PROGRAM StringHelper
VAR
END_VAR

// Converts the provided string to all lower case and returns the converted value.
METHOD ToLowerCase : T_MaxString
VAR_INPUT
	str	: Tc2_System.T_MaxString;	// Source string
END_VAR
ToLowerCase := Tc2_Utilities.F_ToLCase(in := str);
END_METHOD

// Converts the provided string to all upper case and returns the converted value.
METHOD ToUpperCase : Tc2_System.T_MaxString
VAR_INPUT
	str	: Tc2_System.T_MaxString;	// Source string
END_VAR
ToUpperCase := Tc2_Utilities.F_ToUCase(in := str);
END_METHOD

// Removes leading spaces from the character string and returns the reduced character string
METHOD PUBLIC TrimLeftSide : Tc2_System.T_MaxString
VAR_INPUT
	str	: Tc2_System.T_MaxString; // String to be trimmed
END_VAR
TrimRightSide := Tc2_Utilities.F_LTrim(in := str);
END_METHOD

// Truncates all trailing spaces from the specified value and returns the result.
METHOD PUBLIC TrimRightSide : Tc2_System.T_MaxString
VAR_INPUT
	str	: Tc2_System.T_MaxString;	// String to be trimmed
END_VAR
TrimRightSide := Tc2_Utilities.F_RTrim(in := str);
END_METHOD

END_PROGRAM

(* stored: Version 1.1.0.1, ProductVersion 3.1.4024.13
   POU StringHelper: Id {6038c506-8015-0cf2-2085-30a677155028}, SpecialFunc None
   Method ToLowerCase: Id {04af86ff-c3c4-0ee5-29da-879b8d09b6b9}
   Method ToUpperCase: Id {a9f90e08-f042-0b48-3d37-79d4dbe88971}
   Method TrimLeftSide: Id {aaf318c8-56f7-0f39-3b6b-023f532313ad}
   Method TrimRightSide: Id {76095d0f-b051-05a8-3966-5a98e10f20ea} *)
